# EPICS substitutions: ek9000App/Db/EL3041.substitutions
file EL3041.template
{       pattern
        {
                TERMINAL,

        }
        {
        }
}
